TYPE ST_HMIManual :
STRUCT
	
END_STRUCT
END_TYPE

(* stored: Version 1.1.0.1, ProductVersion 3.1.4024.12
   DUT ST_HMIManual: Id {11a85b5a-74c5-4e96-a25c-2799b2639b00} *)
